(* CODESYS project triggers_RECOVERED_2026-08-08T15-33-00.project

Project tree, tasks and I/O mapping:
  Device : CODESYS Control Win V3 x64, CODESYS, version 3.5.22.30
    application Application
      libraries: Standard, 3.5.22.0 (System)
      task MainTask (cyclic, interval t#20ms, priority 1) calls PLC_PRG
      task VISU_TASK (cyclic, interval 100 ms, priority 31) calls VisuElems.Visu_Prg
      visualisation Visualization
      program PLC_PRG [LD]
  text list GlobalTextList
*)

// Device/Application/PLC_PRG
PROGRAM PLC_PRG
VAR
	enable: BOOL;
	i: INT;
	sum: INT;
END_VAR

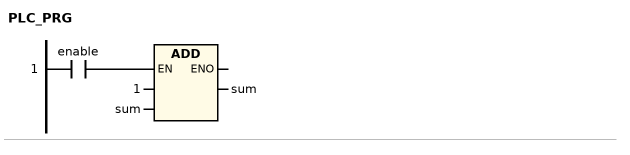
// NETWORK 1
IF enable THEN sum := 1 + sum; END_IF

END_PROGRAM

// Device/Application/Visualization
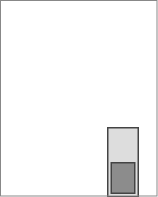
VISUALIZATION Visualization  // 158x197
    DipSwitch (88,127 70x70), variable: PLC_PRG.enable, behaviour: TOGGLE, style: Switch-DipSwitch-Gray
END_VISUALIZATION
